{attribute 'reflection'} 
FUNCTION_BLOCK ABSTRACT FB_GENERAL
VAR //General
  	{attribute 'instance-path'} 
    {attribute 'noinit'} 
	strInstancePath: 	STRING;
END_VAR

METHOD M_CyclicRun : BOOL
VAR_INPUT
END_VAR
END_METHOD

PROPERTY P_ObjectID : STRING
GET
P_ObjectID:='dfknhkljsfa';
END_GET
SET
END_SET
END_PROPERTY

END_FUNCTION_BLOCK

(* stored: Version 1.1.0.1, ProductVersion 3.1.4024.12
   POU FB_GENERAL: Id {c97d6e42-6c96-4c1c-a564-ea2119f54c99}, SpecialFunc None
   Method M_CyclicRun: Id {42bfa581-9cc4-4832-8e5c-44c71c72d56c}
   Property P_ObjectID: Id {c655d5f7-3de4-4711-85be-44f7c9e83db6}
   Get Get: Id {6a3f64e5-0ca4-4354-bdc8-ca2da0767282}
   Set Set: Id {bfee68a6-d97a-4a19-be18-ee462e215d8e} *)
